// SIMATIC S7-200 project (STEP 7-Micro/WIN), CPU 226XM REL 01.22

SYMBOL_TABLE 输入输出
M2               Q0.1     // 拧盖电机
M3               Q0.2     // 瓶盖电机
M5               Q0.5     // 输送带
YV1              Q1.1     // 送盖阀
HL11             Q1.3     // 卡瓶
HL12             Q1.4     // 过载
HL13             Q1.5     // 加盖
HL14             Q1.6     // 无盖
SQ1              I0.0     // 盖检测上限
SQ2              I0.1     // 盖检测下限
SQ3              I0.2     // 进瓶故障
SQ4              I0.3     // 卡瓶
SQ5              I0.4     // 有瓶检测
SQ6              I0.5     // 送盖到位
SA0M             I1.2     // 手动
SA0A             I1.3     // 自动
SA2              I1.5     // 拧盖电机
SA3              I1.6     // 瓶盖电机
SA5              I2.1     // 输送带
SBE              I2.2     // 急停
UF2              I2.3     // 变频故障
QF35             I2.4     // 断路器过载
END_SYMBOL_TABLE

ORGANIZATION_BLOCK MAIN:OB1
TITLE=玻璃瓶压盖机控制程序。设备在实际场景中安装于流水线末端，负责接收灌装完成的瓶子，通过输送带将瓶子送至拧盖位置，依靠拧盖电机完成拧盖动作，并通过瓶盖电机和送盖阀供给瓶盖。
// 
// 在手动模式下，操作员通过控制面板上的拧盖电机开关启动拧盖电机和送盖阀，手动完成拧盖和送盖动作；通过瓶盖电机开关启动瓶盖电机供给瓶盖；通过输送带开关启动输送带移动瓶子。这种模式适用于设备调试或小批量生产。若急停按钮按下时，需确保拧盖电机、瓶盖电机、输送带和送盖阀停止运行，以保障安全。急停按钮用于在紧急情况下暂停设备运行，以保护操作员。
// 
// 在自动模式下，系统通过传感器实现智能化运行。当有瓶检测传感器检测到瓶子到达时，送盖阀打开；当送盖到位传感器触发且无瓶子时，送盖阀关闭。拧盖电机在拧盖电机开关置位，且卡瓶指示灯、过载指示灯和无盖指示灯未点亮时启动。瓶盖电机在瓶盖电机开关置位且盖检测上限传感器未触发时，经过50个时间单位延时后启动；当盖检测上限传感器触发时，经过80个时间单位延时后停止。
// 输送带由输送带开关控制，且需在无卡瓶指示灯和过载指示灯点亮时运行。异常情况通过指示灯提示：卡瓶指示灯在卡瓶检测传感器触发时点亮，过载指示灯在变频故障信号或断路器过载信号触发时点亮，加盖指示灯在加盖检测传感器确认加盖成功时点亮，无盖指示灯在盖检测下限传感器检测到瓶盖不足后延时50个时间单位点亮。
BEGIN
Network 1 // 网络标题
// 网络注释
LDN    SA0M:I1.2
CALL   手动:SBR0
?000
Network 2
LD     SA0A:I1.3
A      SBE:I2.2
CALL   自动:SBR1
?000
Network 3 // 急停
LDN    SA0M:I1.2
AN     SA0M:I1.2
ON     SBE:I2.2
MOVD   0, QD0
Network 4 // 卡瓶
LD     SQ4:I0.3
=      HL11:Q1.3
Network 5 // 过载灯
LD     UF2:I2.3
O      QF35:I2.4
=      HL12:Q1.4
Network 6 // 加盖灯
LD     SQ3:I0.2
=      HL13:Q1.5
Network 7 // 无盖灯
LD     SQ2:I0.1
TON    T103, +50
A      T103
=      HL14:Q1.6
END_ORGANIZATION_BLOCK

SUBROUTINE_BLOCK 手动:SBR0
TITLE=子例行程序注释
BEGIN
Network 1 // 网络标题
// 网络注释
LD     SA2:I1.5
=      M2:Q0.1
=      YV1:Q1.1
Network 2 // 网络标题
// 网络注释
LD     SA3:I1.6
=      M3:Q0.2
Network 3 // 网络标题
// 网络注释
LD     SA5:I2.1
=      M5:Q0.5
Network 4 // 网络标题
// 网络注释
END_SUBROUTINE_BLOCK

SUBROUTINE_BLOCK 自动:SBR1
TITLE=子例行程序注释
BEGIN
Network 1 // 拧盖电机
// 网络注释
LD     SA2:I1.5
AN     HL11:Q1.3
AN     HL12:Q1.4
AN     HL14:Q1.6
=      M2:Q0.1
Network 2 // 瓶盖电机
// 网络注释
LD     SA3:I1.6
LPS
AN     SQ1:I0.0
TON    T101, +50
A      T101
S      M3:Q0.2, 1
LPP
A      SQ1:I0.0
TON    T102, +80
A      T102
R      M3:Q0.2, 1
Network 3
LDN    SA3:I1.6
R      M3:Q0.2, 1
Network 4 // 输送带
// 网络注释
LD     SA5:I2.1
=      M5:Q0.5
Network 5 // 送盖阀
LD     SQ5:I0.4
S      YV1:Q1.1, 1
Network 6
LD     SQ6:I0.5
AN     SQ5:I0.4
R      YV1:Q1.1, 1
Network 7
LD     SQ6:I0.5
EU
SHRB   SQ5:I0.4, M0.0, +4
END_SUBROUTINE_BLOCK
